
(* ===== HMI "HMI_RT_1" =====

HMI tags "EdgeReportTags"
   "rpc_request" : Array [0..100] of WString[254], internal
   "rpc_response" : WString[254], internal
   "TriggerTag1" : Bool, internal
   "rpc_request_status" : Int, internal
   "TemplateFilenameTag" : WString[254], internal
   "ReportStartTimeTag" : WString[254], internal
   "ReportEndTimeTag" : WString[254], internal
   "ReportFilenameTag" : WString[254], internal
   "TriggerDeleteReports" : Bool, internal
*)